Staubli VAL3: remSetMaxV.pgx

program remSetMaxV(string& sArgs[] (dimensions=1), string& sReturn[] (dimensions=1))
  local num bOk
  local num nVal
begin
  // Set the maximum allowed translational velocity in mm/s.
  //
  logMsg("call remSetMaxV")
  call remSetnGlobal(sArgs,nMaxVelo,0,200,"SETMAXV",sReturn)
end
